TYPE ST_AxisDescription :
STRUCT
	iGroupNumber : INT;
    sUnits : STRING := UNIT_mm;
END_STRUCT
END_TYPE

(* stored: Version 1.1.0.1, ProductVersion 3.1.4024.11
   DUT ST_AxisDescription: Id {50ff6038-4325-4846-892a-422b31e6a32f} *)
